{attribute 'qualified_only'}
{attribute 'strict'}
TYPE E_ADC_AXES_ID :
(
	ALL_AXES := 0,
	ADC_1,
	ADC_2
);
END_TYPE

(* stored: Version 1.1.0.1, ProductVersion 3.1.4022.12
   DUT E_ADC_AXES_ID: Id {c0bd9687-ba38-4a20-b43f-ddc6bbd58a08} *)
